ORGANIZATION_BLOCK "Main"
{ S7_Optimized_Access := 'TRUE' }

BEGIN

"FB_Test_DB"();

END_ORGANIZATION_BLOCK
